// TIA Portal V17 export
// export: Created 2022-03-11T11:27:36.1676076Z, ExportSetting WithDefaults, DisplayName Totally Integrated Automation Portal, DisplayVersion V17, DisplayName TIA Portal Openness, DisplayVersion V17, DisplayName TIA Portal Version Control Interface, DisplayVersion V17, DisplayName STEP 7 Professional, DisplayVersion V17, DisplayName STEP 7 Safety, DisplayVersion V17, DisplayName WinCC Advanced, DisplayVersion V17
FUNCTION "ROBNAME" : Void   // FC71, LAD
{ S7_Optimized_Access := 'TRUE' }
VERSION : 1.1
// stored: AutoNumber true, IsIECCheckEnabled false, SetENOAutomatically false, StructureModified 2017-06-20T14:56:00.5916118Z, UDAEnableTagReadback false
   VAR_TEMP
      Temp : Struct
         _Bool : Bool;
         _Byte : Byte;
         _Word : Word;
         _DWord : DWord;
         _Int : Int;
         _DInt : DInt;
         _Real : Real;
         _S5Time : S5Time;
         _Time : Time;
      END_STRUCT;
   END_VAR
BEGIN
END_FUNCTION
